FUNCTION_BLOCK Motor
VAR_INPUT
	//Software
	Stopped : BOOL;
	TurningClockwise : BOOL;
	TurningCounterclockwise : BOOL;
END_VAR
VAR_OUTPUT	
	AI_Position AT %I*: UINT;
	AI_Speed AT %I*: UDINT;
END_VAR
VAR	
	//Hardware
	DO_TurnClockwise AT %Q* : BOOL;
	DO_TurnCounterclockwise AT %Q* : BOOL;	
END_VAR

ACTION ACT_Stop:
DO_TurnClockwise := FALSE;
DO_TurnCounterclockwise := FALSE;

Stopped := TRUE;
TurningClockwise := FALSE;
TurningCounterclockwise := FALSE;
END_ACTION

ACTION ACT_TurnClockwise:
DO_TurnClockwise := TRUE;
DO_TurnCounterclockwise := FALSE;

Stopped := FALSE;
TurningClockwise := TRUE;
TurningCounterclockwise := FALSE;
END_ACTION

ACTION ACT_TurnCounterclockwise:
DO_TurnClockwise := FALSE;
DO_TurnCounterclockwise := TRUE;

Stopped := FALSE;
TurningClockwise := FALSE;
TurningCounterclockwise := TRUE;
END_ACTION

END_FUNCTION_BLOCK

(* stored: Version 1.1.0.1, ProductVersion 3.1.4024.9
   POU Motor: Id {ee44e2ee-d826-40c4-ac13-843b90c8794b}, SpecialFunc None
   Action ACT_Stop: Id {df50afe2-ff71-425b-b230-addf35d47a00}
   Action ACT_TurnClockwise: Id {e9d7b57d-e1ec-4de7-b569-680da77cb241}
   Action ACT_TurnCounterclockwise: Id {ab24c744-b90e-4f1d-a0c6-609a85a904c3} *)
